Fanuc KAREL source: kt00473.KL

PROGRAM KT00473
%STACKSIZE=65535
%PRIORITY=65535
%NOLOCKGROUP
VAR
P1 : POSITION
P2 : POSITION
OUT : BOOLEAN
BEGIN
-- UNRESOLVED_PC line 8 opcodes [49 49 AC 23] marker_code=0
END KT00473
